FUNCTION Convert_DT_TO_UINT : BOOL
VAR_INPUT
	in : DT;
	out : REFERENCE TO UINT;
END_VAR
VAR
	converted : UINT;
END_VAR

converted := DT_TO_UINT(in);

IF (UINT_TO_DT(converted) <> in) THEN
	RETURN;
END_IF

out := converted;
Convert_DT_TO_UINT := TRUE;

END_FUNCTION

(* stored: Version 1.1.0.1, ProductVersion 3.1.4024.12
   POU Convert_DT_TO_UINT: Id {5457aa37-5322-49b7-9232-44bdbbd511c3}, SpecialFunc None *)
